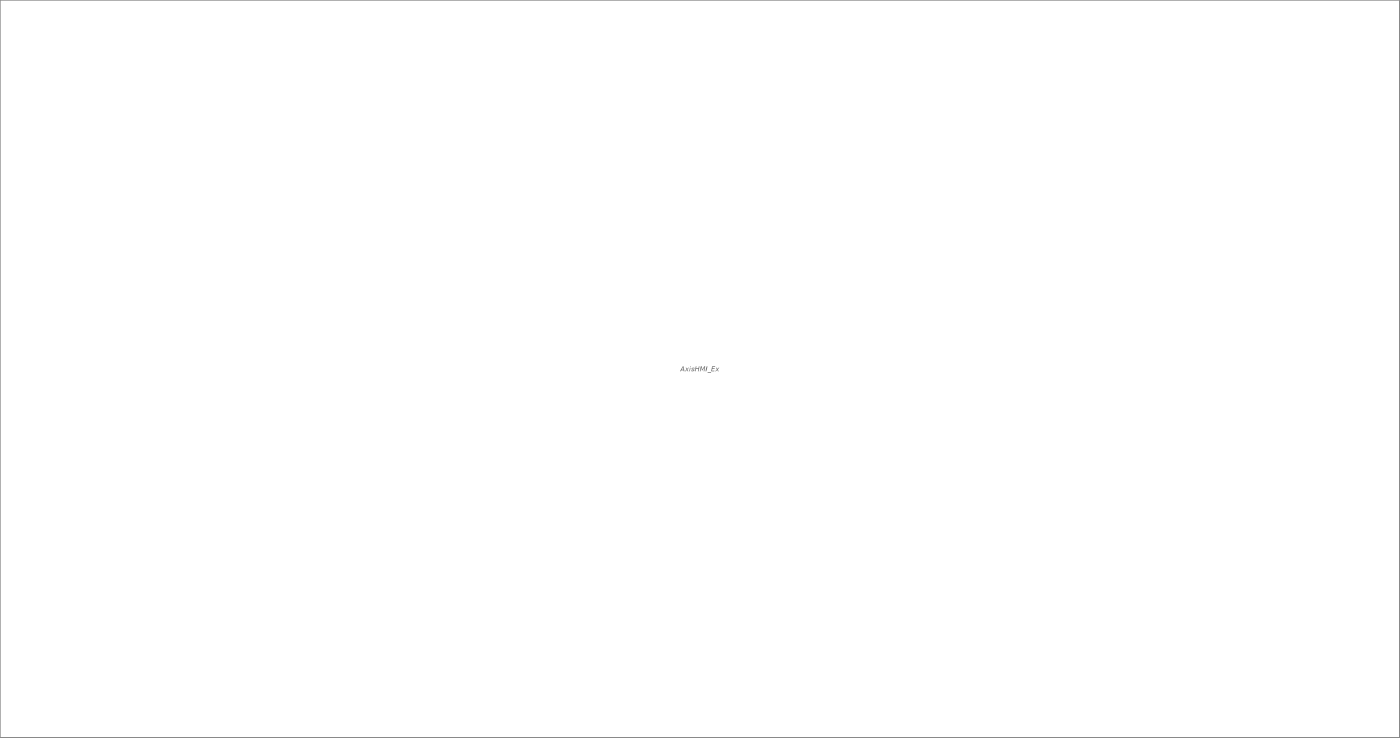
VISUALIZATION visu_FR  // 2048x1080
    TabControl (0,0 2048x1080)
        shows AxisHMI_Ex(stAxisHMI := GVL.fr[G_HMI.iFr].st_mcAxis, mcAxis := GVL.fr[G_HMI.iFr].mcAxis, xError := GVL.fr[G_HMI.iFr].mcAxis.xError)
        shows v_IO_FR(dIO_FR := GVL.fr[G_HMI.iFr])
        shows Axis_HMI(st_axis_HMI := st_mcAxis[EN_Axis.Grip_axis])
        shows v_IO_LC()
        shows v_lc(dIO_LC := GVL.lc[1])
        [0]: TabTitle=FR_axis
        [6]: TabTitle=Gripper
        [1]: AxisHMI=gantrybase.st_mcAxis[EN_Axis.Y], mcAxis=gantrybase.mcAxis[EN_Axis.Y], Error=gantrybase.mcAxis[EN_Axis.Y].xError
        [2]: AxisHMI=gantrybase.st_mcAxis[EN_Axis.Z], mcAxis=gantrybase.mcAxis[EN_Axis.Z], Error=gantrybase.mcAxis[EN_Axis.Z].xError
        p699000190: gantrybase.st_mcAxis[EN_Axis.X]
        p2837713833: gantrybase.mcAxis[EN_Axis.Z].sAxisName
        p520277221: gantrybase.mcAxis[EN_Axis.X].xError
        p3331604638: gantrybase.st_mcAxis[EN_Axis.Z]
        p1813558639: gantrybase.mcAxis[EN_Axis.Z].xError
        p1563495665: gantrybase.st_mcAxis[EN_Axis.Y]
        p2070126892: gantrybase.mcAxis[EN_Axis.Y].xError
        p3435970784: gantrybase.mcAxis[EN_Axis.X]
        p2829954345: gantrybase.mcAxis[EN_Axis.Y]
        p3218520426: gantrybase.mcAxis[EN_Axis.Z]
        p4285860315: GVL.rem[G_HMI.iReM]
        p1681814995: GVL.lc[0]
END_VISUALIZATION

(* stored: Version 1.1.0.1, ProductVersion 3.1.4024.12
   Visu visu_FR: Id {39ce09fc-fb55-4ead-a928-ae197be4d750} *)
